(* IEC 61131-3 sources: test_fernando/Modicon_M660C.device.xml.v3^/Plc Logic.plclogic.xml.v3^/Application.application.xml.v3^, 2 files *)

(* ---- GVL.gvl ---- *)
{attribute 'qualified_only'}
VAR_GLOBAL
END_VAR

(* ---- SR_Main.prg.st ---- *)
PROGRAM SR_Main
VAR
	stTime: DWORD;
	presult: SysTimeRtc.RTS_IEC_RESULT;
	myDate: DATE;
	myTime: TIME;
	myDateTime: DATE_AND_TIME;
	mySetDateTime: DATE_AND_TIME;

	setTime: BOOL;

	iVar: INT;

END_VAR

(*
stTime := SysTimeRtc.SysTimeRtcGet(presult);
myDate := DWORD_TO_DATE(stTime);
myTime := DWORD_TO_TIME(stTime);
myDateTime := DWORD_TO_DT(stTime);

IF setTime THEN
	setTime := FALSE;
	resultSet := sysTimeRtc.SysTimeRtcSet(DT_TO_DWORD(mySetDateTime));
END_IF
*)

iVar := 10;
